PROGRAM Task_1
VAR
	fbDoorControl : FB_DoorControl;   // Instance of the door control function block
	bCardPresented: BOOL;
	bAccessGranted: BOOL;
END_VAR

// Card validation and access granting logic
IF bCardPresented THEN
    bAccessGranted := TRUE;           // Grant access if card is presented
    fbDoorControl(bStartTimer := TRUE);
ELSE
    bAccessGranted := FALSE;
    fbDoorControl(bStartTimer := FALSE);
END_IF

// Write the door status to the GVL
GVL.bDoorClosed := fbDoorControl.bDoorClosed;

END_PROGRAM

(* stored: Version 1.1.0.1, ProductVersion 3.1.4024.12
   POU Task_1: Id {96115f30-6e23-4ae0-a3f5-a348a2e84b6a}, SpecialFunc None *)
